# EPICS alarm handler configuration: mps_database/bareTest/alarms/areas/mpln_feeh_mp01.alhConfig
GROUP NULL MPLN:FEEH:MP01:1
$ALIAS MPS Link Node 145
$GUIDANCE
LTUH MPS
   Group Name: MPLN:FEEH:MP01:1
   Summary PV:  MPLN:FEEH:MP01:1:STATSUMY
$END
CHANNEL  MPLN:FEEH:MP01:1    MPLN:FEEH:MP01:1:MPS_EN_RBV		-----
CHANNEL  MPLN:FEEH:MP01:1    MPLN:FEEH:MP01:1:LC1_MODE_RBV		-----
